FUNCTION_BLOCK T_CallMethod IMPLEMENTS I_Executable
VAR
   logger : I_Logger;
	_symbolHandle : ST_SymbolHandle;
	readWrite : T_AdsReadWrite;
END_VAR
VAR CONSTANT
   LOG_DEBUG : DWORD := 0;
   LOG_INFO : DWORD := ADSLOG_MSGTYPE_HINT;
   LOG_WARNING : DWORD := ADSLOG_MSGTYPE_WARN;
   LOG_ERROR : DWORD := ADSLOG_MSGTYPE_ERROR;
END_VAR

readWrite();

PROPERTY Busy : BOOL
GET
Busy := readWrite.Busy;
END_GET
END_PROPERTY

PROPERTY Done : BOOL
GET
Done := readWrite.Done;
END_GET
END_PROPERTY

PROPERTY Error : BOOL
GET
Error := readWrite.Error;
END_GET
END_PROPERTY

METHOD PRIVATE ToLog
VAR_INPUT
	Msg : STRING(255);
	LogLevel : DWORD; // generic level, can be mapped to logging framework
END_VAR
IF logger = 0 THEN
	RETURN;
	
END_IF

logger.ToLog(Msg, LogLevel);
END_METHOD

METHOD TryMethodCall : BOOL
VAR_INPUT
	symbolHandle : ST_SymbolHandle;
	adsTimeout : TIME := DEFAULT_ADS_TIMEOUT; // DEFAULT_ADS_TIMEOUT is T#5s;
END_VAR
VAR_OUTPUT
	status : I_Executable;
END_VAR
VAR
	readWriteOpts : ST_AdsReadWriteOptions;
END_VAR
VAR CONSTANT
	NO_HANDLE : DWORD := 0;
END_VAR
IF Busy THEN
	ToLog('Cannot TryGetHandle as Busy', LOG_WARNING);
	RETURN;
	
END_IF

_symbolHandle := symbolHandle;

readWriteOpts.AdsAddress := _symbolHandle.SymbolAddress.Ads;
readWriteOpts.IndexGroup := ADSIGRP_SYM_VALBYHND;
readWriteOpts.IndexOffset := _symbolHandle.Handle;
readWriteOpts.WriteParams := _symbolHandle.SymbolAddress.WriteRef;
readWriteOpts.ReadParams := _symbolHandle.SymbolAddress.ReadRef;
readWriteOpts.Timeout := adsTimeout;

TryMethodCall := readWrite.TryRequest( readWriteOpts, status => status );
END_METHOD

END_FUNCTION_BLOCK

(* stored: Version 1.1.0.1, ProductVersion 3.1.4024.9
   POU T_CallMethod: Id {43800a14-cbe5-47c9-ba5a-eb02060ebed4}, SpecialFunc None
   Property Busy: Id {00f364d3-e3a9-4967-95e6-1c1273ef761d}
   Get Get: Id {3cc2f5ee-80f1-46ef-a98e-ca6f7b4788a8}
   Property Done: Id {66e95090-ae94-44d6-9141-353d329f353c}
   Get Get: Id {deeec7ee-ebb3-461e-aa30-9faef40c15a0}
   Property Error: Id {49de12f0-b759-46c8-aa4c-1bf190915d3d}
   Get Get: Id {d5507bf0-9222-4a97-9da5-1cbd64e191c4}
   Method ToLog: Id {0937adbe-d5e3-4e76-944f-dcf1f4b30465}
   Method TryMethodCall: Id {5e373b87-5ead-4214-80c5-acfc0021609b} *)
